{attribute addProperty BoxType "AT2041-0250-0018"}
{attribute addProperty Id "A_0104_AT2042_5250_0019_AT2042_5250AT2042_3DCFC8D064080"}
{attribute addProperty CRC "314151005"}
{attribute addProperty SizeInBites "640"}
{attribute addProperty SizeInBytes "80"}
TYPE A_0040_AT2041_0250_0018_12B9905D EXTENDS AT2041_9506A482 :
STRUCT
	{attribute addProperty Name "A_0104_AT2042_5250_0019_AT2042_5250"}
	A_0104_AT2042_5250_0019_AT2042_5250 : AT2042_3DCFC8D0;
END_STRUCT
END_TYPE

(* stored: Version 1.2.0.0, ProductVersion 3.1.4024.9
   DUT A_0040_AT2041_0250_0018_12B9905D: Id {9dec2879-6f6b-4706-bb59-b16b47a5c887} *)
